SUBAPPLICATION F_AI_RAW_TO_PERCENT_AD (* Volladapterbasierte Alternative zu F_AI_RAW_TO_PERCENT: Analog-Rohwert (AD-Adapter, DWORD 0-4095) linear in Prozent (AR-Adapter, REAL 0.0-100.0) umrechnen, gleiches Ergebnis wie die datenbasierte Variante. WICHTIG: AD_TO_AR/F_DWORD_TO_REAL waere hier FALSCH - das ist eine Bit-Reinterpretation (IEEE754-Cast), keine numerische Umwandlung (siehe forte_real.cpp CIEC_REAL::setValue, case e_DWORD: setValueSimple). Der korrekte Weg ist AD_TO_AUDI (Bit-Reinterpretation DWORD-UDINT, hier gueltig, gleiche Bitbreite/Darstellung) gefolgt von AUDI_TO_AR (nutzt intern F_UDINT_TO_REAL, echte numerische Umwandlung). *)
  (* Standard: 61499-2 *)
  (* Version 1.0, 2026-08-30, franz *)
  PACKAGE MyLib::sys;
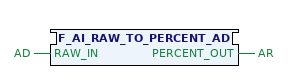
  SOCKETS
    RAW_IN : adapter::types::unidirectional::AD; (* Analog-Rohwert 0-4095 (12 bit, logiBUS_AI_IDA.IN) *)
  END_SOCKETS
  PLUGS
    PERCENT_OUT : adapter::types::unidirectional::AR; (* Prozent 0.0-100.0, linear raw/4095*100, keine physikalische Einheit *)
  END_PLUGS
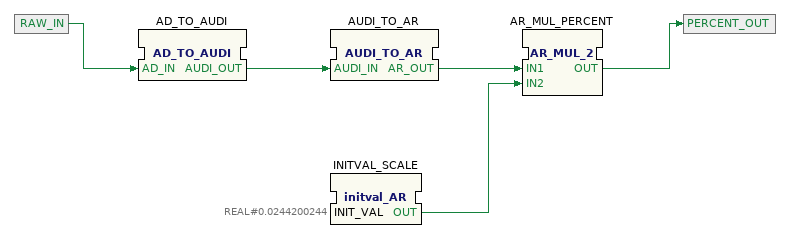
  FBS
    AD_TO_AUDI : adapter::conversion::unidirectional::AD_TO_AUDI;
    AUDI_TO_AR : adapter::conversion::unidirectional::AUDI_TO_AR;
    INITVAL_SCALE : adapter::types::unidirectional::AR::initval::initval_AR(INIT_VAL := REAL#0.0244200244);
    AR_MUL_PERCENT : adapter::iec61131::arithmetic::AR_MUL_2;
  END_FBS
  ADAPTER_CONNECTIONS
    RAW_IN TO AD_TO_AUDI.AD_IN;
    AD_TO_AUDI.AUDI_OUT TO AUDI_TO_AR.AUDI_IN;
    AUDI_TO_AR.AR_OUT TO AR_MUL_PERCENT.IN1;
    INITVAL_SCALE.OUT TO AR_MUL_PERCENT.IN2;
    AR_MUL_PERCENT.OUT TO PERCENT_OUT;
  END_CONNECTIONS
END_SUBAPPLICATION
